# EPICS StreamDevice protocol: protocols/anatrg.proto
Terminator = LF;
ExtraInput = Ignore;
ReplyTimeout = 2500;

setAnaTrg {
	out "anatrg_\$2 -H %(\$1:H.RVAL)d -- %(\$1:M)s %(\$1:L1.RVAL)d %(\$1:L2.RVAL)d";
	in;
}

setAnaTrgOr {
	out "atd_OR %(\$1:1)04x%(\$1:0)04x";
	in;
}

setAnaTrgAnd {
	out "atd_AND %(\$1:1)04x%(\$1:0)04x";
	in;
}

getAnaTrgSrc {
	out "status_latch";
	in "%(\$1)x,%x";
}

setAnaTrgGroupMask {
	out "group_trigger_mask %(\$1:1)04x,%(\$1:2)04x";
	in;
}

getAnaTrgGroupStatus {
	out "group_status_latch";
	in "%(\$1)04x,%04x";
}

set_group_status_mode {
	out "group_status_mode %d";
	in;
}

get_group_status_mode {
	out "group_status_mode";
	in "%d";
}

set_group_first_n {
	out "group_first_n_triggers %d";
	in;
}

setAnaTrgScale {
	out "ATD_CSR.SHL %(RVAL)d";
	in;
}

setAnaTrgSpad {
	out "ATD_CSR.SPAD_ON %d";
	in;
}
setDelTrg {
	out "deltrg_\$1 %d";
	in;
}

setDelZN {
	out "dtd_ZN 0x%x";
	in;
}

setATD_Reset {
	out "ATD_CSR.ATD_RESET %d";
	in;
}
